FUNCTION_BLOCK FB_RoutingStation EXTENDS FB_XPlanarStationBase
VAR_INPUT
END_VAR
VAR_OUTPUT
END_VAR
VAR
	_OutputA	: I_XplanarStation;
	_OutputB	: I_XPlanarStation;
END_VAR

METHOD Execute
SUPER^.Execute(); //Call the base station logic to handle sending and receiving of movers

//When the station is in the Process mover state you can perform any application specific station logic
IF StationState = E_XPlanarStationState.ProcessMover THEN
	IF _OutputA <> 0 AND _OutputB <> 0 THEN	
		CASE ipCurrentMover.MoverIndex OF
			1, 3:
				ipNextStation := _OutputA;
			2, 4:
				ipNextStation := _OutputB;
		END_CASE
		
		_StationComplete := TRUE;	//Set _StationComplete TRUE when done.  This will be automatically reset when the mover exits
	END_IF
END_IF
END_METHOD

PROPERTY OutputA : I_XPlanarStation
SET
_OutputA := OutputA;
END_SET
END_PROPERTY

PROPERTY OutputB : I_XPlanarStation
SET
_OutputB := OutputB;
END_SET
END_PROPERTY

END_FUNCTION_BLOCK

(* stored: Version 1.1.0.1, ProductVersion 3.1.4024.13
   POU FB_RoutingStation: Id {d1f931ac-72f8-4dc5-a0d5-c8a34bfee707}, SpecialFunc None
   Method Execute: Id {317fc10b-70df-4800-b6e1-124d9fdfd392}
   Property OutputA: Id {199a749e-f95a-4b6d-a7fb-62cd714a449b}
   Set Set: Id {a3c98b37-a790-4d7e-a53f-902f71112374}
   Property OutputB: Id {714b125d-edd6-456f-b213-a30f84db27fa}
   Set Set: Id {d22e7d3e-ca00-4e41-a66f-0b6a0816a096} *)
